Universal Robots PolyScope program: remote_control.urp

Program remote_control (installation=default directory=/programs createdIn=3.2.19275.0 lastSavedIn=5.4.0.76181 robotSerialNumber=20195500451)
Calibrated DH parameters: a=[0.00002, -0.231658, -0.317125, 0.000011, 0.000055, 0]; d=[0.162082, 123.190176, -180.284242, 57.22734, 0.099524, 0.09934]; alpha=[1.569304, 0.00289, 0.004025, 1.569925, -1.569026, 0]; deltaTheta=[0, 0.993923, 4.662183, 0.627072, 0.000001, 0]
BeforeStart
  setq := [0,0,0,0,0,0]
  selection_vec := [0,0,0,0,0,0]
  wrench := [0,0,0,0,0,0]
  limits := [0,0,0,0,0,0]
  ctrl_type := 0
  blocking := 0.008
  lookahead := 0.03
  gain := 500
  maxPosError := 0.01
  maxOrientError := 0.01
  Script: zero_ftsensor()
Robot Program (runOnlyOnce=false)
  If ctrl_type == 1
    Script: servoj(setq,0,0,blocking,lookahead,gain)
  ElseIf ctrl_type == 2
    Script: speedj(setq,gain,blocking)
  ElseIf ctrl_type == 3
    Script: movej(setq,gain,maxPosError,blocking,maxOrientError)
  ElseIf ctrl_type == 4
    Script: movel(setq,gain,maxPosError,blocking,maxOrientError)
  ElseIf ctrl_type == 5
    Script: force_mode(Base,selection_vec,wrench,2,limits)
  Script: sync()
Thread Thread_1 (runOnlyOnce=false trackProgramExecution=false)
  Folder Read remote registers
    tmp := [0,0,0,0,0,0,0,0,0,0,0,0]
    Script: tmp[0] = read_input_float_register(0)
    Script: tmp[1] = read_input_float_register(1)
    Script: tmp[2] = read_input_float_register(2)
    Script: tmp[3] = read_input_float_register(3)
    Script: tmp[4] = read_input_float_register(4)
    Script: tmp[5] = read_input_float_register(5)
    Script: tmp[6] = read_input_float_register(6)
    Script: tmp[7] = read_input_float_register(7)
    Script: tmp[8] = read_input_float_register(8)
    Script: tmp[9] = read_input_float_register(9)
    Script: tmp[10] = read_input_float_register(10)
    Script: tmp[11] = read_input_float_register(11)
  If tmp != [0,0,0,0,0,0,0,0,0,0,0,0]
    If ctrl_type ≥1 and ctrl_type≤4
      setq := [tmp[0],tmp[1],tmp[2],tmp[3],tmp[4],tmp[5]]
      ctrl_type := tmp[6]
      blocking := tmp[7]
      lookahead := tmp[8]
      gain := tmp[9]
      maxPosError := tmp[10]
      maxOrientError := tmp[11]
    ElseIf ctrl_type == 5
      wrench := [tmp[0],tmp[1],tmp[2],tmp[3],tmp[4],tmp[5]]
      selection_vec := [tmp[6],tmp[7],tmp[8],tmp[9],tmp[10],tmp[11]]
      limits := [tmp[12],tmp[13],tmp[14],tmp[15],tmp[16],tmp[17]]
  Script: sync()
Thread Thread_2 (runOnlyOnce=false trackProgramExecution=false)
  Folder Send Torque Values
    torque := get_joint_torques()
    Script: write_output_float_register(0, torque[0])
    Script: write_output_float_register(1, torque[1])
    Script: write_output_float_register(2, torque[2])
    Script: write_output_float_register(3, torque[3])
    Script: write_output_float_register(4, torque[4])
    Script: write_output_float_register(5, torque[5])
